// TIA Portal V20 export
// export: Created 2025-12-01T14:56:14.8881008Z, ExportSetting None, DisplayName Totally Integrated Automation Portal, DisplayVersion V20 Update 3, DisplayName TIA Portal Openness, DisplayVersion V20 Update 3, DisplayName TIA Portal Version Control Interface, DisplayVersion V20 Update 3, DisplayName STEP 7 Professional, DisplayVersion V20 Update 3, DisplayName STEP 7 Safety, DisplayVersion V20 Update 2, DisplayName WinCC Basic/Comfort/Advanced, DisplayVersion V20 Update 3, DisplayName WinCC Professional, DisplayVersion V20 Update 3, DisplayName WinCC Unified, DisplayVersion V20 Update 3
TYPE "ROUT_Datos_Pantalla_Scanner"
   STRUCT
      Numero_Mesa : Int := 0;
      Diagnostico : Struct
         Device_Ready : Bool := FALSE;
         System_Ready : Bool := FALSE;
         Good_Read : Bool := FALSE;
         No_Read : Bool := FALSE;
         External_output_1 : Bool := FALSE;
         External_output_2 : Bool := FALSE;
         Result_1 : Bool := FALSE;
         Result_2 : Bool := FALSE;
         External_input_1 : Bool := FALSE;
         External_input_2 : Bool := FALSE;
         Sensor_1 : Bool := FALSE;
         Sensor_2 : Bool := FALSE;
         Definable_1 : Bool := FALSE;
         Definable_2 : Bool := FALSE;
         Definable_3 : Bool := FALSE;
         Definable_4 : Bool := FALSE;
      END_STRUCT;
      errores : Struct
         lecturas_consecuti : Bool := FALSE;
         porcentaje : Bool := FALSE;
         Error_reserva1 : Bool := FALSE;
         Error_reserva2 : Bool := FALSE;
         Error_reserva3 : Bool := FALSE;
         Error_reserva4 : Bool := FALSE;
         Error_reserva5 : Bool := FALSE;
         Error_reserva6 : Bool := FALSE;
         Error_reserva7 : Bool := FALSE;
         Error_reserva8 : Bool := FALSE;
         Error_reserva9 : Bool := FALSE;
         Error_reserva10 : Bool := FALSE;
         Error_reserva11 : Bool := FALSE;
         Error_reserva12 : Bool := FALSE;
         Error_reserva13 : Bool := FALSE;
         Error_scanner : Bool := FALSE;
      END_STRUCT;
      Lectura : Array[0..31] of Char;
      contadores { S7_SetPoint := 'True'} : "ROUT_Estadisticas_Scanners";
      orden_pantalla : Struct
         disparo : Bool := FALSE;
         reset : Bool := FALSE;
         RESERVA_1 : Bool := FALSE;
         RESERVA_2 : Bool := FALSE;
         RESERVA_3 : Bool := FALSE;
         RESERVA_4 : Bool := FALSE;
         RESERVA_5 : Bool := FALSE;
         RESERVA_6 : Bool := FALSE;
         RESERVA_7 : Bool := FALSE;
         RESERVA_8 : Bool := FALSE;
         RESERVA_9 : Bool := FALSE;
         RESERVA_10 : Bool := FALSE;
         RESERVA_11 : Bool := FALSE;
         RESERVA_12 : Bool := FALSE;
         RESERVA_13 : Bool := FALSE;
         RESERVA_14 : Bool := FALSE;
      END_STRUCT;
   END_STRUCT;
END_TYPE
